// TIA Portal V21 export
TYPE "OBJ_Washing_Recipe_v100_Type"
   STRUCT
      "i_Index Limit" : Int;   // Qty of Step on This Recipe
      "i_Pos End Recipe" : Int;   // Last Step of Washing Recipe
      DW0 : Int;   // Timer accumulator
      DW1 : Int;   // Counter Pitch Accumulator
      DW2 : Int;   // Container Counter Accumulator
      DW3 : Int;
      DW4 : Int;
      DW5 : Int;   // Inlet Temperature>Set Point Temperature
      DW6 : Int;   // Inlet Temperature<Set Point Temperature
      DW7 : Int;   // Hopper Temperature>Set Point Temperature
      DW8 : Int;   // Hopper Temperature<Set Point Temperature
      DW9 : Int;   // Volume > Set Point Volume
      DW10 : Int;   // Volume < Set Point Volume
      DW11 : Int;   // Filler position
      DW12 : Int;
      DW13 : Int;
      DW14 : Int;   // Input State 1
      DW15 : Int;   // Input State 2
      DW16 : Int;
      DW17 : Int;
      DW18 : Int;
      DW19 : Int;
      DW20 : Int;
      DW21 : Int := 16;
      DW22 : Int;
      DW23 : Int;
      "@_StepOnWork" { S7_SetPoint := 'True'} : "OBJ_Washing_Step_V210_Type";
      DW31 : Int;   // Function Step
      DW32 : Int := 10;
      DW33 : Word;
      DW34 : Word;   // Visualizzo il set point del numero di cicli di FLIP FLOP
      DW35 : Word;
      DW36 : Int;
      DW37 : DWord;
      DW39 : DWord;
      DW41 : Word;
      DW42 : Int := 110;
      DW43 : Word;
      DW44 : Word;
      DW45 : Word;
      DW46 : DInt;
      DW48 : Word;
      i_Type_Of_Wash : Int;
      "@_Step" { S7_SetPoint := 'True'} : Array[0..100] of "OBJ_Washing_Step_V210_Type";
   END_STRUCT;
END_TYPE
